RoboDK station: Stringer B-Top3-BOX1.rdk

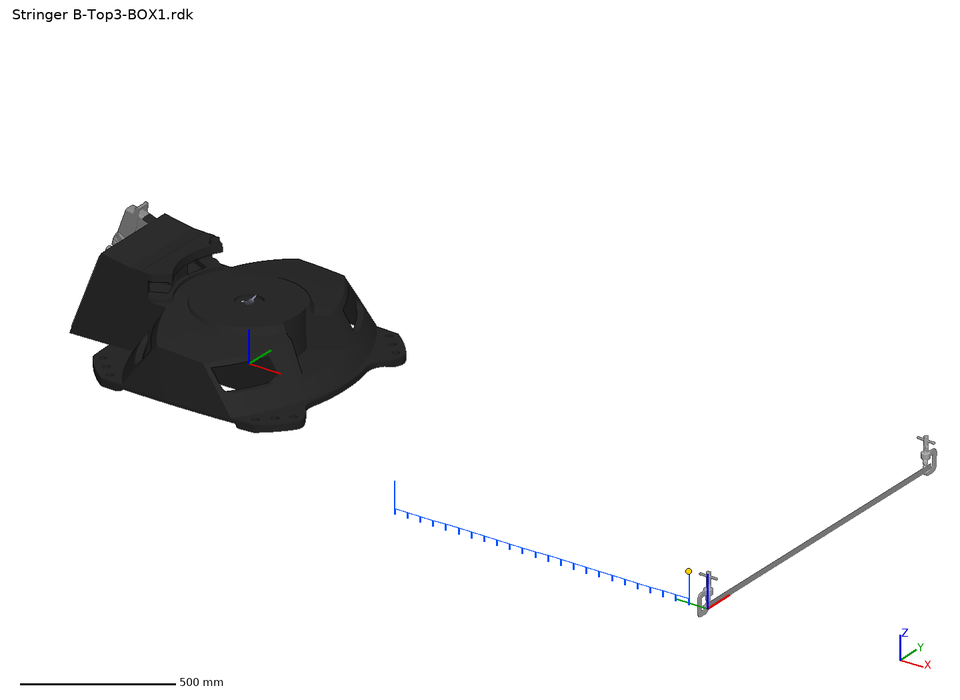
[picture v0: the station drawn from its stored meshes, robots at their saved joint values, targets as dots, program paths as lines]
Station Stringer B-Top3-BOX1 (saved by RoboDK 5.2.3). Poses are relative to the parent item; angles as X-Y-Z fixed-axis rotations.
  - frame KUKA KR 210 R2700 extra Base at (0, 0, 0) mm
    - robot KUKA KR 210 R2700 extra: 6 axes, payload 210 kg, reach 2696 mm, repeatability 0.06 mm, weight 1068 kg
        joint limits [-185, -140, -120, -350, -125, -350] to [185, -5, 155, 350, 125, 350]; home [0, -90, 90, 0, 0, 0]; saved at [-38.862, -26.822, 86.576, 94.614, 23.337, -127.078]
      - tool Spindle, TCP at (32, 0, 260) mm, rotated rx 0 ry 39 rz 0 deg, size 157.3 x 72 x 259.9 mm
  - frame Frame 2 at (1800, 0, -372.68) mm, rotated rx 0 ry 0 rz 90 deg
    - object L-Stringer B - Top3-BOX1 at (0, 0, 0) mm, size 1250 x 20 x 20 mm, geometry from L-Stringer B - Top3-BOX1.stl
    - object Stringer B-Top3-BOX1 at (0, 0, 0) mm, rotated rx 0 ry 0 rz -90 deg, 24 curves, geometry from Point 24
  - machining project Point settings: rotZ(0) | rotX(0)*rotY(0) | rotz(0) | onStart | onPathStart | onApproach | onPoint | onRetract | onFinish | SetRPM(%1) | SetTool(%1) | Extruder(%1) | default | default | OutOnMov(%1) | OutOffMov(%1) | onPathFinish | M_RunCode(%1)
  - program Point (131 instructions, listed below)
  - object FinalClamp at (1789.91, 16.41, -309.43) mm, rotated rx 35.23 ry 89.37 rz -143.56 deg, size 145.3 x 71.1 x 72 mm, geometry from FinalClamp.stp
  - object FinalClamp2 at (1789.66, 1236.1, -310.01) mm, rotated rx 180 ry 88.27 rz 180 deg, size 145.3 x 71.1 x 72 mm, geometry from FinalClamp.stp
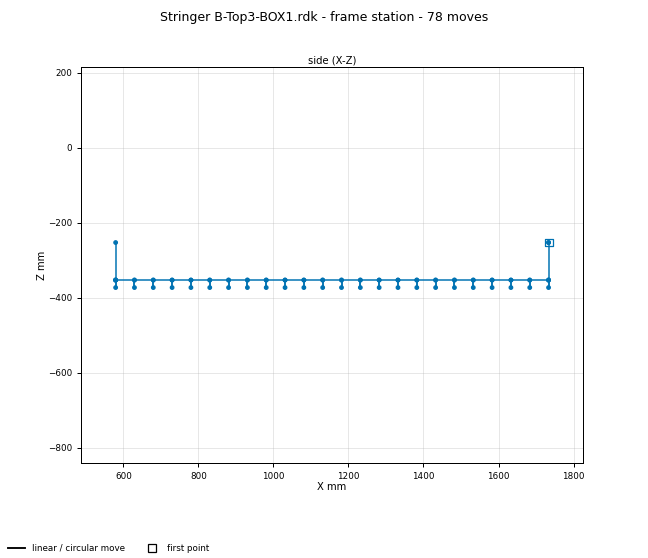
[picture p0: tool path of Stringer B-Top3-BOX1.rdk in frame station, 78 of 78 moves have a stored position in this frame; points joined in program order, loops and branches not executed]

--- program Point (robot KUKA KR 210 R2700 extra) ---
  Smooth(1)
  Set speed (1000.0 mm/s)
  Set Ref.: Frame 2
  Set Tool: Spindle
  Show Spindle
  MoveJ 1 to (-11.2, 66.57, 120) mm, rotated rx 180 ry 0 rz -180 deg; joints [-2.516, -34.012, 111.84, 176.492, 26.844, -178.825]
  MoveL 2 to (-11.2, 66.57, 120) mm, rotated rx 180 ry 0 rz -180 deg; joints [-2.516, -34.012, 111.84, 176.492, 26.844, -178.825]
  MoveL 3 to (-11.2, 66.57, 20) mm, rotated rx -180 ry 0 rz -180 deg; joints [-2.516, -28.683, 109.197, 176.786, 29.526, -179.159]
  MoveL 4 to (-11.2, 66.57, 20) mm, rotated rx -180 ry 0 rz -180 deg; joints [-2.516, -28.683, 109.197, 176.786, 29.526, -179.159]
  Set speed (50.0 mm/s)
  MoveL 5 to (-11.2, 66.57, 0) mm, rotated rx 180 ry 0 rz 180 deg; joints [-2.516, -27.625, 108.621, 176.833, 30.007, -179.213]
  MoveL 6 to (-11.2, 66.57, 20) mm, rotated rx -180 ry 0 rz -180 deg; joints [-2.516, -28.683, 109.197, 176.786, 29.526, -179.159]
  Set speed (1000.0 mm/s)
  MoveL 7 to (-11.2, 116.75, 20) mm, rotated rx -180 ry 0 rz -180 deg; joints [-4.407, -28.661, 109.04, 174.349, 29.415, -178.501]
  Set speed (50.0 mm/s)
  MoveL 8 to (-11.2, 116.75, 0) mm, rotated rx -180 ry 0 rz -180 deg; joints [-4.407, -27.605, 108.464, 174.431, 29.894, -178.596]
  MoveL 9 to (-11.2, 116.75, 20) mm, rotated rx -180 ry 0 rz -180 deg; joints [-4.407, -28.661, 109.04, 174.349, 29.415, -178.501]
  Set speed (1000.0 mm/s)
  MoveL 10 to (-11.2, 166.92, 20) mm, rotated rx -180 ry 0 rz -180 deg; joints [-6.288, -28.627, 108.796, 171.889, 29.245, -177.806]
  Set speed (50.0 mm/s)
  MoveL 11 to (-11.2, 166.92, 0) mm, rotated rx 180 ry 0 rz 180 deg; joints [-6.288, -27.573, 108.222, 172.008, 29.72, -177.943]
  MoveL 12 to (-11.2, 166.92, 20) mm, rotated rx -180 ry 0 rz -180 deg; joints [-6.288, -28.627, 108.796, 171.889, 29.245, -177.806]
  Set speed (1000.0 mm/s)
  MoveL 13 to (-11.2, 217.09, 20) mm, rotated rx 180 ry 0 rz -180 deg; joints [-8.156, -28.581, 108.467, 169.394, 29.019, -177.056]
  Set speed (50.0 mm/s)
  MoveL 14 to (-11.2, 217.09, 0) mm, rotated rx -180 ry 0 rz -180 deg; joints [-8.156, -27.529, 107.894, 169.55, 29.489, -177.235]
  MoveL 15 to (-11.2, 217.09, 20) mm, rotated rx 180 ry 0 rz -180 deg; joints [-8.156, -28.581, 108.467, 169.394, 29.019, -177.056]
  Set speed (1000.0 mm/s)
  MoveL 16 to (-11.2, 267.27, 20) mm, rotated rx 180 ry 0 rz -180 deg; joints [-10.007, -28.52, 108.053, 166.855, 28.741, -176.236]
  Set speed (50.0 mm/s)
  MoveL 17 to (-11.2, 267.27, 0) mm, rotated rx -180 ry 0 rz -180 deg; joints [-10.007, -27.472, 107.481, 167.049, 29.204, -176.458]
  MoveL 18 to (-11.2, 267.27, 20) mm, rotated rx 180 ry 0 rz -180 deg; joints [-10.007, -28.52, 108.053, 166.855, 28.741, -176.236]
  Set speed (1000.0 mm/s)
  MoveL 19 to (-11.2, 317.44, 20) mm, rotated rx 180 ry 0 rz 180 deg; joints [-11.836, -28.443, 107.553, 164.261, 28.415, -175.329]
  Set speed (50.0 mm/s)
  MoveL 20 to (-11.2, 317.44, 0) mm, rotated rx 180 ry 0 rz 180 deg; joints [-11.836, -27.4, 106.983, 164.494, 28.871, -175.595]
  MoveL 21 to (-11.2, 317.44, 20) mm, rotated rx 180 ry 0 rz 180 deg; joints [-11.836, -28.443, 107.553, 164.261, 28.415, -175.329]
  Set speed (1000.0 mm/s)
  MoveL 22 to (-11.2, 367.62, 20) mm, rotated rx 180 ry 0 rz 180 deg; joints [-13.642, -28.35, 106.967, 161.599, 28.047, -174.319]
  Set speed (50.0 mm/s)
  MoveL 23 to (-11.2, 367.62, 0) mm, rotated rx 180 ry 0 rz 180 deg; joints [-13.642, -27.312, 106.4, 161.873, 28.494, -174.63]
  MoveL 24 to (-11.2, 367.62, 20) mm, rotated rx 180 ry 0 rz 180 deg; joints [-13.642, -28.35, 106.967, 161.599, 28.047, -174.319]
  Set speed (1000.0 mm/s)
  MoveL 25 to (-11.2, 417.79, 20) mm, rotated rx -180 ry 0 rz -180 deg; joints [-15.42, -28.239, 106.298, 158.86, 27.644, -173.19]
  Set speed (50.0 mm/s)
  MoveL 26 to (-11.2, 417.79, 0) mm, rotated rx -180 ry 0 rz -180 deg; joints [-15.42, -27.206, 105.732, 159.176, 28.079, -173.548]
  MoveL 27 to (-11.2, 417.79, 20) mm, rotated rx -180 ry 0 rz -180 deg; joints [-15.42, -28.239, 106.298, 158.86, 27.644, -173.19]
  Set speed (1000.0 mm/s)
  MoveL 28 to (-11.2, 467.96, 20) mm, rotated rx 180 ry 0 rz 180 deg; joints [-17.168, -28.107, 105.544, 156.032, 27.211, -171.929]
  Set speed (50.0 mm/s)
  MoveL 29 to (-11.2, 467.96, 0) mm, rotated rx 180 ry 0 rz -180 deg; joints [-17.168, -27.081, 104.981, 156.392, 27.635, -172.334]
  MoveL 30 to (-11.2, 467.96, 20) mm, rotated rx 180 ry 0 rz 180 deg; joints [-17.168, -28.107, 105.544, 156.032, 27.211, -171.929]
  Set speed (1000.0 mm/s)
  MoveL 31 to (-11.2, 518.14, 20) mm, rotated rx 180 ry 0 rz -180 deg; joints [-18.884, -27.953, 104.706, 153.102, 26.758, -170.518]
  Set speed (50.0 mm/s)
  MoveL 32 to (-11.2, 518.14, 0) mm, rotated rx 180 ry 0 rz 180 deg; joints [-18.884, -26.934, 104.145, 153.507, 27.168, -170.972]
  MoveL 33 to (-11.2, 518.14, 20) mm, rotated rx 180 ry 0 rz -180 deg; joints [-18.884, -27.953, 104.706, 153.102, 26.758, -170.518]
  Set speed (1000.0 mm/s)
  MoveL 34 to (-11.2, 568.31, 20) mm, rotated rx -180 ry 0 rz -180 deg; joints [-20.565, -27.776, 103.784, 150.061, 26.292, -168.946]
  Set speed (50.0 mm/s)
  MoveL 35 to (-11.2, 568.31, 0) mm, rotated rx 180 ry 0 rz 180 deg; joints [-20.565, -26.764, 103.226, 150.512, 26.686, -169.45]
  MoveL 36 to (-11.2, 568.31, 20) mm, rotated rx -180 ry 0 rz -180 deg; joints [-20.565, -27.776, 103.784, 150.061, 26.292, -168.946]
  Set speed (1000.0 mm/s)
  MoveL 37 to (-11.2, 618.49, 20) mm, rotated rx 180 ry 0 rz 180 deg; joints [-22.211, -27.572, 102.779, 146.897, 25.823, -167.198]
  Set speed (50.0 mm/s)
  MoveL 38 to (-11.2, 618.49, 0) mm, rotated rx -180 ry 0 rz -180 deg; joints [-22.211, -26.568, 102.223, 147.396, 26.199, -167.753]
  MoveL 39 to (-11.2, 618.49, 20) mm, rotated rx 180 ry 0 rz 180 deg; joints [-22.211, -27.572, 102.779, 146.897, 25.823, -167.198]
  Set speed (1000.0 mm/s)
  MoveL 40 to (-11.2, 668.66, 20) mm, rotated rx 180 ry 0 rz 180 deg; joints [-23.818, -27.341, 101.691, 143.602, 25.359, -165.265]
  Set speed (50.0 mm/s)
  MoveL 41 to (-11.2, 668.66, 0) mm, rotated rx -180 ry 0 rz -180 deg; joints [-23.818, -26.345, 101.138, 144.149, 25.717, -165.87]
  MoveL 42 to (-11.2, 668.66, 20) mm, rotated rx 180 ry 0 rz 180 deg; joints [-23.818, -27.341, 101.691, 143.602, 25.359, -165.265]
  Set speed (1000.0 mm/s)
  MoveL 43 to (-11.2, 718.83, 20) mm, rotated rx 180 ry 0 rz 180 deg; joints [-25.387, -27.08, 100.52, 140.168, 24.912, -163.136]
  Set speed (50.0 mm/s)
  MoveL 44 to (-11.2, 718.83, 0) mm, rotated rx 180 ry 0 rz -180 deg; joints [-25.387, -26.092, 99.969, 140.762, 25.249, -163.792]
  MoveL 45 to (-11.2, 718.83, 20) mm, rotated rx 180 ry 0 rz 180 deg; joints [-25.387, -27.08, 100.52, 140.168, 24.912, -163.136]
  Set speed (1000.0 mm/s)
  MoveL 46 to (-11.2, 769.01, 20) mm, rotated rx -180 ry 0 rz -180 deg; joints [-26.916, -26.787, 99.265, 136.589, 24.491, -160.806]
  Set speed (50.0 mm/s)
  MoveL 47 to (-11.2, 769.01, 0) mm, rotated rx -180 ry 0 rz -180 deg; joints [-26.916, -25.808, 98.717, 137.23, 24.805, -161.512]
  MoveL 48 to (-11.2, 769.01, 20) mm, rotated rx -180 ry 0 rz -180 deg; joints [-26.916, -26.787, 99.265, 136.589, 24.491, -160.806]
  Set speed (1000.0 mm/s)
  MoveL 49 to (-11.2, 819.18, 20) mm, rotated rx -180 ry 0 rz 180 deg; joints [-28.405, -26.46, 97.928, 132.865, 24.107, -158.273]
  Set speed (50.0 mm/s)
  MoveL 50 to (-11.2, 819.18, 0) mm, rotated rx -180 ry 0 rz -180 deg; joints [-28.405, -25.49, 97.382, 133.551, 24.397, -159.026]
  MoveL 51 to (-11.2, 819.18, 20) mm, rotated rx -180 ry 0 rz 180 deg; joints [-28.405, -26.46, 97.928, 132.865, 24.107, -158.273]
  Set speed (1000.0 mm/s)
  MoveL 52 to (-11.2, 869.35, 20) mm, rotated rx 180 ry 0 rz -180 deg; joints [-29.853, -26.097, 96.507, 128.997, 23.77, -155.539]
  Set speed (50.0 mm/s)
  MoveL 53 to (-11.2, 869.35, 0) mm, rotated rx 180 ry 0 rz -180 deg; joints [-29.853, -25.137, 95.963, 129.724, 24.035, -156.334]
  MoveL 54 to (-11.2, 869.35, 20) mm, rotated rx 180 ry 0 rz -180 deg; joints [-29.853, -26.097, 96.507, 128.997, 23.77, -155.539]
  Set speed (1000.0 mm/s)
  MoveL 55 to (-11.2, 919.53, 20) mm, rotated rx 180 ry 0 rz -180 deg; joints [-31.26, -25.697, 95.001, 124.991, 23.492, -152.609]
  Set speed (50.0 mm/s)
  MoveL 56 to (-11.2, 919.53, 0) mm, rotated rx 180 ry 0 rz -180 deg; joints [-31.26, -24.746, 94.459, 125.755, 23.729, -153.443]
  MoveL 57 to (-11.2, 919.53, 20) mm, rotated rx 180 ry 0 rz -180 deg; joints [-31.26, -25.697, 95.001, 124.991, 23.492, -152.609]
  Set speed (1000.0 mm/s)
  MoveL 58 to (-11.2, 969.7, 20) mm, rotated rx 180 ry 0 rz 180 deg; joints [-32.626, -25.257, 93.411, 120.863, 23.283, -149.498]
  Set speed (50.0 mm/s)
  MoveL 59 to (-11.2, 969.7, 0) mm, rotated rx 180 ry 0 rz -180 deg; joints [-32.626, -24.315, 92.871, 121.657, 23.492, -150.363]
  MoveL 60 to (-11.2, 969.7, 20) mm, rotated rx 180 ry 0 rz 180 deg; joints [-32.626, -25.257, 93.411, 120.863, 23.283, -149.498]
  Set speed (1000.0 mm/s)
  MoveL 61 to (-11.2, 1019.88, 20) mm, rotated rx -180 ry 0 rz -180 deg; joints [-33.953, -24.775, 91.734, 116.627, 23.152, -146.223]
  Set speed (50.0 mm/s)
  MoveL 62 to (-11.2, 1019.88, 0) mm, rotated rx -180 ry 0 rz -180 deg; joints [-33.953, -23.843, 91.195, 117.443, 23.331, -147.111]
  MoveL 63 to (-11.2, 1019.88, 20) mm, rotated rx -180 ry 0 rz -180 deg; joints [-33.953, -24.775, 91.734, 116.627, 23.152, -146.223]
  Set speed (1000.0 mm/s)
  MoveL 64 to (-11.2, 1070.05, 20) mm, rotated rx 180 ry 0 rz -180 deg; joints [-35.238, -24.25, 89.971, 112.31, 23.109, -142.809]
  Set speed (50.0 mm/s)
  MoveL 65 to (-11.2, 1070.05, 0) mm, rotated rx 180 ry 0 rz 180 deg; joints [-35.238, -23.326, 89.432, 113.139, 23.258, -143.712]
  MoveL 66 to (-11.2, 1070.05, 20) mm, rotated rx 180 ry 0 rz -180 deg; joints [-35.238, -24.25, 89.971, 112.31, 23.109, -142.809]
  Set speed (1000.0 mm/s)
  MoveL 67 to (-11.2, 1120.22, 20) mm, rotated rx -180 ry 0 rz -180 deg; joints [-36.485, -23.678, 88.117, 107.939, 23.161, -139.286]
  Set speed (50.0 mm/s)
  MoveL 68 to (-11.2, 1120.22, 0) mm, rotated rx -180 ry 0 rz -180 deg; joints [-36.485, -22.764, 87.579, 108.771, 23.28, -140.192]
  MoveL 69 to (-11.2, 1120.22, 20) mm, rotated rx -180 ry 0 rz -180 deg; joints [-36.485, -23.678, 88.117, 107.939, 23.161, -139.286]
  Set speed (1000.0 mm/s)
  MoveL 70 to (-11.2, 1170.4, 20) mm, rotated rx -180 ry 0 rz -180 deg; joints [-37.692, -23.059, 86.172, 103.546, 23.315, -135.684]
  Set speed (50.0 mm/s)
  MoveL 71 to (-11.2, 1170.4, 0) mm, rotated rx -180 ry 0 rz -180 deg; joints [-37.692, -22.153, 85.633, 104.371, 23.404, -136.583]
  MoveL 72 to (-11.2, 1170.4, 20) mm, rotated rx -180 ry 0 rz -180 deg; joints [-37.692, -23.059, 86.172, 103.546, 23.315, -135.684]
  Set speed (1000.0 mm/s)
  MoveL 73 to (-11.2, 1220.57, 20) mm, rotated rx -180 ry 0 rz -180 deg; joints [-38.862, -22.388, 84.132, 99.166, 23.576, -132.041]
  Set speed (50.0 mm/s)
  MoveL 74 to (-11.2, 1220.57, 0) mm, rotated rx 180 ry 0 rz 180 deg; joints [-38.862, -21.491, 83.592, 99.973, 23.636, -132.921]
  MoveL 75 to (-11.2, 1220.57, 20) mm, rotated rx -180 ry 0 rz -180 deg; joints [-38.862, -22.388, 84.132, 99.166, 23.576, -132.041]
  MoveL 76 to (-11.2, 1220.57, 20) mm, rotated rx -180 ry 0 rz -180 deg; joints [-38.862, -22.388, 84.132, 99.166, 23.576, -132.041]
  Set speed (1000.0 mm/s)
  MoveL 77 to (-11.2, 1220.57, 20) mm, rotated rx -180 ry 0 rz -180 deg; joints [-38.862, -22.388, 84.132, 99.166, 23.576, -132.041]
  MoveL 78 to (-11.2, 1220.57, 120) mm, rotated rx 180 ry 0 rz 180 deg; joints [-38.862, -26.822, 86.576, 94.614, 23.337, -127.078]
